# EPICS substitutions: iocBoot/ioc13Hytec/DAC.substitutions
file "$(DAC128V)/dac128VApp/Db/singleDAC.db"
{
pattern
{P,        D, N, C,  PORT,  S,  EGUL,  DRVL,  LOPR, EGUF, DRVH, HOPR, PREC, LINR,  VAL}

# Set all channels to read in V and have full +-10V range
{13Hytec:, 1, 1, 0,  DAC1,  0, -10.0,  -10.,  -10.,   10.,  10,  10,    3,  LINEAR, 0.0}
{13Hytec:, 1, 2, 0,  DAC1,  1, -10.0,  -10.,  -10.,   10.,  10,  10,    3,  LINEAR, 0.0}
{13Hytec:, 1, 3, 0,  DAC1,  2, -10.0,  -10.,  -10.,   10.,  10,  10,    3,  LINEAR, 0.0}
{13Hytec:, 1, 4, 0,  DAC1,  3, -10.0,  -10.,  -10.,   10.,  10,  10,    3,  LINEAR, 0.0}
{13Hytec:, 1, 5, 0,  DAC1,  4, -10.0,  -10.,  -10.,   10.,  10,  10,    3,  LINEAR, 0.0}
{13Hytec:, 1, 6, 0,  DAC1,  5, -10.0,  -10.,  -10.,   10.,  10,  10,    3,  LINEAR, 0.0}
{13Hytec:, 1, 7, 0,  DAC1,  6, -10.0,  -10.,  -10.,   10.,  10,  10,    3,  LINEAR, 0.0}
{13Hytec:, 1, 8, 0,  DAC1,  7, -10.0,  -10.,  -10.,   10.,  10,  10,    3,  LINEAR, 0.0}
}
